FUNCTION_BLOCK fbSpeech EXTENDS fbSimpleRemoteExec

METHOD  Execute : BOOL
VAR_INPUT
	param : ANY;
END_VAR
Speak(
END_METHOD

METHOD PRIVATE Speak : BOOL
VAR_INPUT
	_sentence : STRING(255);
END_VAR
END_METHOD

END_FUNCTION_BLOCK

(* stored: Version 1.1.0.1, ProductVersion 3.1.4024.3
   POU fbSpeech: Id {1a4b5a0b-3b73-432d-acfd-383a393272b8}, SpecialFunc None
   Method Execute: Id {4512e749-38a3-4d44-b934-bdb29e383b99}
   Method Speak: Id {413cdf48-41a9-4d34-8eb9-9c3890a86ada} *)
